FUNCTION_BLOCK "G303M_Code"
TITLE =G303M LOUVER AIR HEATER KILN 2
//COPYRIGHT:    (C) 2009  BUHLER AG, CH-9240 UZWIL, SWITZERLAND
//
//PRODUCT:      WinCoS_BIW01_09
//
//TITLE:        LOUVER AIR HEATER KILN 2
//                Machine group control
//                Maschinengruppensteuerung
//
//--------------------------------------------------------------------------------
//
//IDENT:        AUTHOR:             DEPT:                              DATE:
//
//P01_FB403.2.0 M.Wedler            AEB41                              27.Apr.2010
//             2nd Release
//P01_FB403.1.0 K.Renz              CSB41                              08.Okt.2009
//             1st Release
//
//--------------------------------------------------------------------------------
//
//PURPOSE:
//
//MANUAL :
//
//RESTRICTIONS:
//
//--------------------------------------------------------------------------------
AUTHOR : KR
FAMILY : USW
VERSION : 9.9


VAR
  Gr : "GCS7_GrpCtrlSub";	//Standard interface to group
  InOutValue1 : DINT ;	//Data for user
  InOutValue2 : DINT ;	//Data for user
  OutWayConflict : BOOL ;	//Data for user
  OutSelectionOk : BOOL ;	//Data for user
  CmdNewValue : BOOL ;	//Data for user
  CmdNewJob : BOOL ;	//Data for user
  OutCodeOK : BOOL ;	//Data for user
  InEndOfJob : BOOL ;	//Data for user
  staWayOk : BOOL ;	//Data for user
  EdgeStartRelease : BOOL ;	//Data for user
  USW8 : BOOL ;	//Data for user
  USW9 : BOOL ;	//Data for user
  USW10 : BOOL ;	//Data for user
  USW11 : BOOL ;	//Data for user
  USW12 : BOOL ;	//Data for user
  USW13 : BOOL ;	//Data for user
  USW14 : BOOL ;	//Data for user
  USW15 : BOOL ;	//Data for user
  A_3240_MXZ11 : "GCS7_E_ValveControl4Pos";	// VLS4Ctrl
  A_3240_MXZ11I1 : "GCS7_E_DigInput";	// DigInpCont
  A_3240_MXZ11I11 : "GCS7_E_DigInput";	// DigInpCont
  A_3240_MXZ11I2 : "GCS7_E_DigInput";	// DigInpCont
  A_3240_MXZ11I22 : "GCS7_E_DigInput";	// DigInpCont
  A_3241_MXZ11 : "GCS7_E_ValveControl4Pos";	// VLS4Ctrl
  A_3241_MXZ11I1 : "GCS7_E_DigInput";	// DigInpCont
  A_3241_MXZ11I11 : "GCS7_E_DigInput";	// DigInpCont
  A_3241_MXZ11I2 : "GCS7_E_DigInput";	// DigInpCont
  A_3241_MXZ11I22 : "GCS7_E_DigInput";	// DigInpCont
END_VAR
VAR_TEMP
  tmpEnable : BOOL ;
  tmpFlag : BOOL ;
  tmpCmdNext : BOOL ;
  tmpLocal : BOOL ;
  tmpAspOk : BOOL ;
  tmpHWStop : BOOL ;
  tmpInstanzDBNo : INT ;
END_VAR
BEGIN
NETWORK
TITLE =



NETWORK
TITLE =Read command from group control
//Parameter
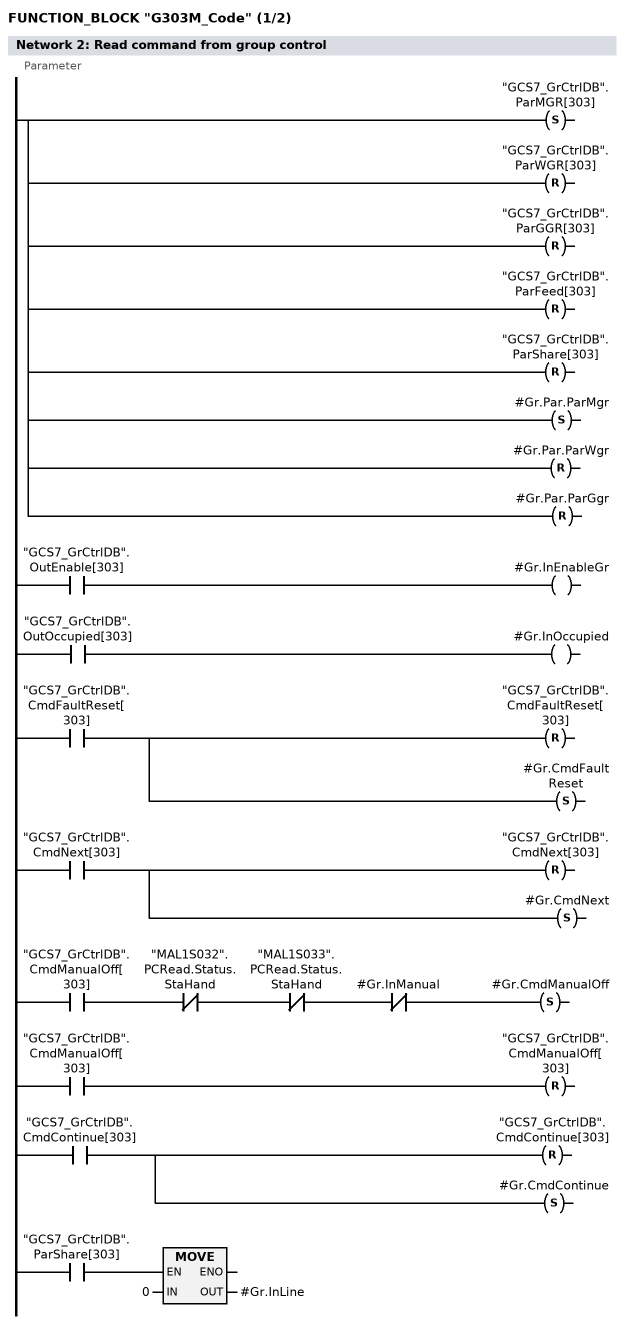
      SET   ;
      S     "GCS7_GrCtrlDB".ParMGR[303];
      R     "GCS7_GrCtrlDB".ParWGR[303];
      R     "GCS7_GrCtrlDB".ParGGR[303];
      R     "GCS7_GrCtrlDB".ParFeed[303];
      R     "GCS7_GrCtrlDB".ParShare[303];
      S     #Gr.Par.ParMgr;
      R     #Gr.Par.ParWgr;
      R     #Gr.Par.ParGgr;
//Command
      U     "GCS7_GrCtrlDB".OutEnable[303];
      =     #Gr.InEnableGr;
      U     "GCS7_GrCtrlDB".OutOccupied[303];
      =     #Gr.InOccupied;
      U     "GCS7_GrCtrlDB".CmdFaultReset[303];
      R     "GCS7_GrCtrlDB".CmdFaultReset[303];
      S     #Gr.CmdFaultReset;
      U     "GCS7_GrCtrlDB".CmdNext[303];
      R     "GCS7_GrCtrlDB".CmdNext[303];
      S     #Gr.CmdNext;

      U     "GCS7_GrCtrlDB".CmdManualOff[303];
      UN    "MAL1S032".PCRead.Status.StaHand;
      UN    "MAL1S033".PCRead.Status.StaHand;
      UN    #Gr.InManual;
      S     #Gr.CmdManualOff;
      U     "GCS7_GrCtrlDB".CmdManualOff[303];
      R     "GCS7_GrCtrlDB".CmdManualOff[303];

//      U     "GCS7_GrCtrlDB".CmdManualOff[303]
//      O     "GCS7_GrCtrlDB".OutOccupied[303]
//      R     "GCS7_GrCtrlDB".CmdManualOff[303]
//      S     #Gr.CmdManualOff

      U     "GCS7_GrCtrlDB".CmdContinue[303];
      R     "GCS7_GrCtrlDB".CmdContinue[303];
      S     #Gr.CmdContinue;
//Init Line Number
      U     "GCS7_GrCtrlDB".ParShare[303];
      SPBN  WE00;
      L     0;
      T     #Gr.InLine;
WE00: NOP   0;
NETWORK
TITLE =Call Methode Control
// 1. Handle Interface PCControl
// 2. Prepare mode --> ModePassive,ModeActive,ModeIdling
// 3. Reset global flags of the group
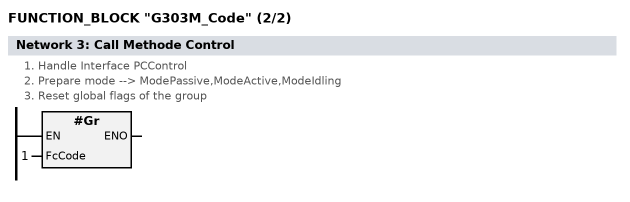
      CALL #Gr (
           FcCode                   := 1);
NETWORK
TITLE =Restart Idling Time

      L     #Gr.Par.ParIdling;
      L     2;
      >=I   ;
      SPB   IdTm;
      T     #Gr.Par.ParIdling;
IdTm: NOP   0;
      U     #A_3240_MXZ11.StNoPosition;
      O     #A_3241_MXZ11.StNoPosition;
      UN    #Gr.InOccupied;
      S     #Gr.CmdRestartIdling;
NETWORK
TITLE =Prepare global flags



NETWORK
TITLE =Set Pattern (Target position)

      L     "MAL1S033Par".Ilo.ILOMode;
      L     5;
      ==I   ;
      U     #Gr.InManual;
      SPBN  M062;
      L     1000;
      T     #A_3240_MXZ11.InPositionMiddle; // setpoint element
      T     #A_3241_MXZ11.InPositionMiddle; // setpoint element
      SPA   M060;
M062: NOP   0;
// setpoint louver air heater
      U     "MAL1S033Par".Par.FlagProcess.ProcessActive;
      UN    "MAL1S033Par".Par.FlagProcess.Cooling_Activ;
      O(    ;
      U     "MAL1S033Par".Par.FlagProcess.Cooling_Activ;
      UN    "G298M".A_3250_MXZ11.StHN;
      UN    "G298M".A_3251_MXZ11.StHN;
      UN    "G298M".A_3252_MXZ11.StHN;
      UN    "G298M".A_3253_MXZ11.StHN;
      )     ;
      SPBN  M061;
      L     1000;
      T     #A_3240_MXZ11.InPositionMiddle; // setpoint element
      T     #A_3241_MXZ11.InPositionMiddle; // setpoint element
M061: NOP   0;
      U(    ;
      U     "MAL1S033Par".Par.FlagProcess.ProcessEnd;
      ON    "MAL1S033Par".Par.FlagProcess.ProcessActive;
      )     ;
      SPBN  M060;
      L     0;
      T     #A_3240_MXZ11.InPositionMiddle; // setpoint element
      T     #A_3241_MXZ11.InPositionMiddle; // setpoint element
M060: NOP   0;

NETWORK
TITLE =Interlocking WayOk



NETWORK
TITLE =Interlocking Autostart

      CLR   ;
      R     #Gr.OutAutostart;
NETWORK
TITLE =Interlocking Enable
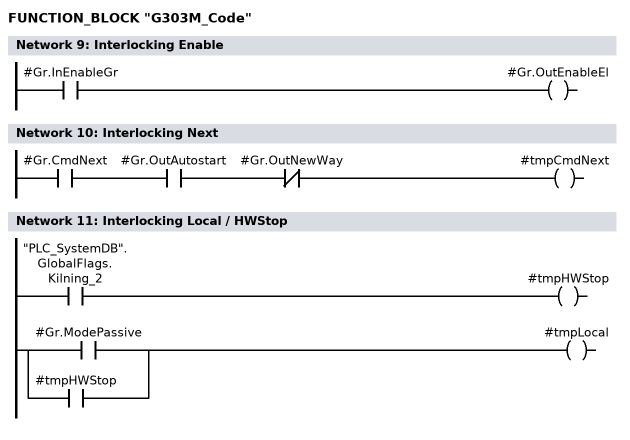

      U     #Gr.InEnableGr;
      =     #Gr.OutEnableEl;

NETWORK
TITLE =Interlocking Next

      U     #Gr.CmdNext;
      U     #Gr.OutAutostart;
      UN    #Gr.OutNewWay;
      =     #tmpCmdNext;

NETWORK
TITLE =Interlocking Local / HWStop

      U     "PLC_SystemDB".GlobalFlags.Kilning_2;
      =     #tmpHWStop;

      U     #Gr.ModePassive;
      O     #tmpHWStop;
      =     #tmpLocal;

NETWORK
TITLE ==A-3240-MXZ11 : LOUVER-AIR ON DOOR FOR RECYCLE AIR 1

      NOP   0;
//-InLocal---
      U(    ;
      U     #tmpLocal;
//      U     #A_3240_MXZ11I11.StTrue
      U     #A_3240_MXZ11.StLN;
      O     ;
      U     #Gr.InManual;
      UN    #Gr.InOutAutostartMan;
      )     ;
      =     #A_3240_MXZ11.InLocal;
//
//-Interlocking---
      U     #A_3240_MXZ11.Par.ParManual;
      U     #A_3240_MXZ11.InManual;
      SPB   man1;
      U(    ;
      UN    #Gr.InOccupied;
      UN    #Gr.InManual;
      )     ;
      O(    ;
      L     0;
      L     #A_3240_MXZ11.InPositionMiddle; // setpoint element
      ==I   ;
      )     ;
      U(    ;
      U     #Gr.InManual;
      U     #Gr.InOutAutostartMan;
      ON    #Gr.InManual;
      )     ;
// Function Added, to get shure always closed in passive state
//      U     #Gr.OutEnableEl
      U(    ;
      U     #Gr.OutEnableEl;
      O     ;
      UN    #Gr.InOccupied;
      UN    #Gr.InManual;
      UN    #A_3240_MXZ11.InLocal;
      )     ;
      =     #A_3240_MXZ11.InLN;

      U(    ;
      L     #A_3240_MXZ11.InPositionMiddle; // setpoint element
      L     0;
      >I    ;
      )     ;
      U(    ;
      L     #A_3240_MXZ11.InPositionMiddle; // setpoint element
      L     1000; // 100,0%
      <I    ;
      )     ;
      U(    ;
      U     #Gr.InManual;
      U     #Gr.InOutAutostartMan;
      ON    #Gr.InManual;
      )     ;
      U     #Gr.OutEnableEl;
      S     #A_3240_MXZ11.CmdMiddle1;

      CLR   ;
      S     #A_3240_MXZ11.CmdMiddle2;

      U(    ;
      L     #A_3240_MXZ11.InPositionMiddle; // setpoint element
      L     1000; // 100,0%
      >=I   ;
      )     ;
      U(    ;
      U     #Gr.InManual;
      U     #Gr.InOutAutostartMan;
      ON    #Gr.InManual;
      )     ;
      U     #Gr.OutEnableEl;
      S     #A_3240_MXZ11.CmdHN;
man1: NOP   0;
//
//-Read inputs---
      U     "A_3240_BZS14_I1";
      =     #A_3240_MXZ11.InpLN;
      CLR   ;
      =     #A_3240_MXZ11.InpMiddle1;
      U     "A_3240_BZS15_I1";
      =     #A_3240_MXZ11.InpHN;
      U     "PLC_SystemDB".GlobalFlags.Kilning_2;
      =     #A_3240_MXZ11.InHWStop;
      U     "PLC_DPInfo".Master[1].SlavesError[101];
      =     #A_3240_MXZ11.InDPFault;
//
//-Set Parameters---
//
//-Call object control---
      CALL #A_3240_MXZ11 ;
//
//-Write outputs---
      U     #A_3240_MXZ11.OutpLN;
      =     "A_3240_MXZ11_O1";
      U     #A_3240_MXZ11.OutpHN;
      =     "A_3240_MXZ11_O2";
NETWORK
TITLE ==A-3240-MXZ11I1 : LOUVER-AIR ON DOOR FOR RECYCLE AIR 1 CLOSING

      NOP   0;
//-InLocal---
      U     #tmpLocal;
      SET   ;
      =     #A_3240_MXZ11I1.InLocal;
//
//-Monitoring---
      U     #A_3240_MXZ11.OutpLN; // closing
      =     #A_3240_MXZ11I1.InMonTrue;
      CLR   ;
      =     #A_3240_MXZ11I1.InMonFalse;
//
//-PreAlarm---
      CLR   ;
      =     #A_3240_MXZ11I1.InPreAlarmTrue;
      CLR   ;
      =     #A_3240_MXZ11I1.InPreAlarmFalse;
//
//-Additional commands---
//      CLR
//      S     #A_3240_MXZ11I1.CmdRunTimeOutTime
//
//-Read inputs---
      U     "A_3240_MXZ11_I1";
      =     #A_3240_MXZ11I1.InpTrue;
      U     "PLC_SystemDB".GlobalFlags.Kilning_2;
      =     #A_3240_MXZ11I1.InHWStop;
      U     "PLC_DPInfo".Master[1].SlavesError[101];
      =     #A_3240_MXZ11I1.InDPFault;
//
//-Set Parameters---
//
//-Call object control---
      CALL #A_3240_MXZ11I1 ;
//
//-Write outputs---
NETWORK
TITLE ==A-3240-MXZ11I11 : LOUVER-AIR ON DOOR FOR RECYCLE AIR 1 CLOSED

      NOP   0;
//-InLocal---
      U     #tmpLocal;
      =     #A_3240_MXZ11I11.InLocal;
//
//-Monitoring---
      CLR   ;
      =     #A_3240_MXZ11I11.InMonTrue;
      CLR   ;
      =     #A_3240_MXZ11I11.InMonFalse;
//
//-PreAlarm---
      CLR   ;
      =     #A_3240_MXZ11I11.InPreAlarmTrue;
      CLR   ;
      =     #A_3240_MXZ11I11.InPreAlarmFalse;
//
//-Additional commands---
//      CLR
//      S     #A_3240_MXZ11I11.CmdRunTimeOutTime
//
//-Read inputs---
      U     "A_3240_MXZ11_I1";
      =     #A_3240_MXZ11I11.InpTrue;
      U     "PLC_SystemDB".GlobalFlags.Kilning_2;
      =     #A_3240_MXZ11I11.InHWStop;
      U     "PLC_DPInfo".Master[1].SlavesError[101];
      =     #A_3240_MXZ11I11.InDPFault;
//
//-Set Parameters---
//
//-Call object control---
      CALL #A_3240_MXZ11I11 ;
//
//-Write outputs---
NETWORK
TITLE ==A-3240-MXZ11I2 : LOUVER-AIR ON DOOR FOR RECYCLE AIR 1 OPENING

      NOP   0;
//-InLocal---
      U     #tmpLocal;
      SET   ;
      =     #A_3240_MXZ11I2.InLocal;
//
//-Monitoring---
      U     #A_3240_MXZ11.OutpHN; // opening
      =     #A_3240_MXZ11I2.InMonTrue;
      CLR   ;
      =     #A_3240_MXZ11I2.InMonFalse;
//
//-PreAlarm---
      CLR   ;
      =     #A_3240_MXZ11I2.InPreAlarmTrue;
      CLR   ;
      =     #A_3240_MXZ11I2.InPreAlarmFalse;
//
//-Additional commands---
//      CLR
//      S     #A_3240_MXZ11I2.CmdRunTimeOutTime
//
//-Read inputs---
      U     "A_3240_MXZ11_I2";
      =     #A_3240_MXZ11I2.InpTrue;
      U     "PLC_SystemDB".GlobalFlags.Kilning_2;
      =     #A_3240_MXZ11I2.InHWStop;
      U     "PLC_DPInfo".Master[1].SlavesError[101];
      =     #A_3240_MXZ11I2.InDPFault;
//
//-Set Parameters---
//
//-Call object control---
      CALL #A_3240_MXZ11I2 ;
//
//-Write outputs---
NETWORK
TITLE ==A-3240-MXZ11I22 : LOUVER-AIR ON DOOR FOR RECYCLE AIR 1 OPENED

      NOP   0;
//-InLocal---
      U     #tmpLocal;
      =     #A_3240_MXZ11I22.InLocal;
//
//-Monitoring---
      CLR   ;
      =     #A_3240_MXZ11I22.InMonTrue;
      CLR   ;
      =     #A_3240_MXZ11I22.InMonFalse;
//
//-PreAlarm---
      CLR   ;
      =     #A_3240_MXZ11I22.InPreAlarmTrue;
      CLR   ;
      =     #A_3240_MXZ11I22.InPreAlarmFalse;
//
//-Additional commands---
//      CLR
//      S     #A_3240_MXZ11I22.CmdRunTimeOutTime
//
//-Read inputs---
      U     "A_3240_MXZ11_I2";
      =     #A_3240_MXZ11I22.InpTrue;
      U     "PLC_SystemDB".GlobalFlags.Kilning_2;
      =     #A_3240_MXZ11I22.InHWStop;
      U     "PLC_DPInfo".Master[1].SlavesError[101];
      =     #A_3240_MXZ11I22.InDPFault;
//
//-Set Parameters---
//
//-Call object control---
      CALL #A_3240_MXZ11I22 ;
//
//-Write outputs---
NETWORK
TITLE ==A-3241-MXZ11 : LOUVER-AIR ON DOOR FOR RECYCLE AIR 2

      NOP   0;
//-InLocal---
      U(    ;
      U     #tmpLocal;
//      U     #A_3241_MXZ11I11.StTrue
      U     #A_3241_MXZ11.StLN;
      O     ;
      U     #Gr.InManual;
      UN    #Gr.InOutAutostartMan;
      )     ;
      =     #A_3241_MXZ11.InLocal;
//
//-Interlocking---
      U     #A_3241_MXZ11.Par.ParManual;
      U     #A_3241_MXZ11.InManual;
      SPB   man2;
      U(    ;
      UN    #Gr.InOccupied;
      UN    #Gr.InManual;
      )     ;
      O(    ;
      L     0;
      L     #A_3241_MXZ11.InPositionMiddle; // setpoint element
      ==I   ;
      )     ;
      U(    ;
      U     #Gr.InManual;
      U     #Gr.InOutAutostartMan;
      ON    #Gr.InManual;
      )     ;
// Function Added, to get shure always closed in passive state
//      U     #Gr.OutEnableEl
      U(    ;
      U     #Gr.OutEnableEl;
      O     ;
      UN    #Gr.InOccupied;
      UN    #Gr.InManual;
      UN    #A_3241_MXZ11.InLocal;
      )     ;
      =     #A_3241_MXZ11.InLN;

      U(    ;
      L     #A_3241_MXZ11.InPositionMiddle; // setpoint element
      L     0;
      >I    ;
      )     ;
      U(    ;
      L     #A_3241_MXZ11.InPositionMiddle; // setpoint element
      L     1000; // 100,0%
      <I    ;
      )     ;
      U(    ;
      U     #Gr.InManual;
      U     #Gr.InOutAutostartMan;
      ON    #Gr.InManual;
      )     ;
      U     #Gr.OutEnableEl;
      S     #A_3241_MXZ11.CmdMiddle1;

      CLR   ;
      S     #A_3241_MXZ11.CmdMiddle2;

      U(    ;
      L     #A_3241_MXZ11.InPositionMiddle; // setpoint element
      L     1000; // 100,0%
      >=I   ;
      )     ;
      U(    ;
      U     #Gr.InManual;
      U     #Gr.InOutAutostartMan;
      ON    #Gr.InManual;
      )     ;
      U     #Gr.OutEnableEl;
      S     #A_3241_MXZ11.CmdHN;
man2: NOP   0;
//
//-Read inputs---
      U     "A_3241_BZS14_I1";
      =     #A_3241_MXZ11.InpLN;
      CLR   ;
      =     #A_3241_MXZ11.InpMiddle1;
      U     "A_3241_BZS15_I1";
      =     #A_3241_MXZ11.InpHN;
      U     "PLC_SystemDB".GlobalFlags.Kilning_2;
      =     #A_3241_MXZ11.InHWStop;
      U     "PLC_DPInfo".Master[1].SlavesError[101];
      =     #A_3241_MXZ11.InDPFault;
//
//-Set Parameters---
//
//-Call object control---
      CALL #A_3241_MXZ11 ;
//
//-Write outputs---
      U     #A_3241_MXZ11.OutpLN;
      =     "A_3241_MXZ11_O1";
      U     #A_3241_MXZ11.OutpHN;
      =     "A_3241_MXZ11_O2";
NETWORK
TITLE ==A-3241-MXZ11I1 : LOUVER-AIR ON DOOR FOR RECYCLE AIR 2 CLOSING

      NOP   0;
//-InLocal---
      U     #tmpLocal;
      SET   ;
      =     #A_3241_MXZ11I1.InLocal;
//
//-Monitoring---
      U     #A_3241_MXZ11.OutpLN; // closing
      =     #A_3241_MXZ11I1.InMonTrue;
      CLR   ;
      =     #A_3241_MXZ11I1.InMonFalse;
//
//-PreAlarm---
      CLR   ;
      =     #A_3241_MXZ11I1.InPreAlarmTrue;
      CLR   ;
      =     #A_3241_MXZ11I1.InPreAlarmFalse;
//
//-Additional commands---
//      CLR
//      S     #A_3241_MXZ11I1.CmdRunTimeOutTime
//
//-Read inputs---
      U     "A_3241_MXZ11_I1";
      =     #A_3241_MXZ11I1.InpTrue;
      U     "PLC_SystemDB".GlobalFlags.Kilning_2;
      =     #A_3241_MXZ11I1.InHWStop;
      U     "PLC_DPInfo".Master[1].SlavesError[101];
      =     #A_3241_MXZ11I1.InDPFault;
//
//-Set Parameters---
//
//-Call object control---
      CALL #A_3241_MXZ11I1 ;
//
//-Write outputs---
NETWORK
TITLE ==A-3241-MXZ11I11 : LOUVER-AIR ON DOOR FOR RECYCLE AIR 2 CLOSED

      NOP   0;
//-InLocal---
      U     #tmpLocal;
      =     #A_3241_MXZ11I11.InLocal;
//
//-Monitoring---
      CLR   ;
      =     #A_3241_MXZ11I11.InMonTrue;
      CLR   ;
      =     #A_3241_MXZ11I11.InMonFalse;
//
//-PreAlarm---
      CLR   ;
      =     #A_3241_MXZ11I11.InPreAlarmTrue;
      CLR   ;
      =     #A_3241_MXZ11I11.InPreAlarmFalse;
//
//-Additional commands---
//      CLR
//      S     #A_3241_MXZ11I11.CmdRunTimeOutTime
//
//-Read inputs---
      U     "A_3241_MXZ11_I1";
      =     #A_3241_MXZ11I11.InpTrue;
      U     "PLC_SystemDB".GlobalFlags.Kilning_2;
      =     #A_3241_MXZ11I11.InHWStop;
      U     "PLC_DPInfo".Master[1].SlavesError[101];
      =     #A_3241_MXZ11I11.InDPFault;
//
//-Set Parameters---
//
//-Call object control---
      CALL #A_3241_MXZ11I11 ;
//
//-Write outputs---
NETWORK
TITLE ==A-3241-MXZ11I2 : LOUVER-AIR ON DOOR FOR RECYCLE AIR 2 OPENING

      NOP   0;
//-InLocal---
      U     #tmpLocal;
      SET   ;
      =     #A_3241_MXZ11I2.InLocal;
//
//-Monitoring---
      U     #A_3241_MXZ11.OutpHN; // opening
      =     #A_3241_MXZ11I2.InMonTrue;
      CLR   ;
      =     #A_3241_MXZ11I2.InMonFalse;
//
//-PreAlarm---
      CLR   ;
      =     #A_3241_MXZ11I2.InPreAlarmTrue;
      CLR   ;
      =     #A_3241_MXZ11I2.InPreAlarmFalse;
//
//-Additional commands---
//      CLR
//      S     #A_3241_MXZ11I2.CmdRunTimeOutTime
//
//-Read inputs---
      U     "A_3241_MXZ11_I2";
      =     #A_3241_MXZ11I2.InpTrue;
      U     "PLC_SystemDB".GlobalFlags.Kilning_2;
      =     #A_3241_MXZ11I2.InHWStop;
      U     "PLC_DPInfo".Master[1].SlavesError[101];
      =     #A_3241_MXZ11I2.InDPFault;
//
//-Set Parameters---
//
//-Call object control---
      CALL #A_3241_MXZ11I2 ;
//
//-Write outputs---
NETWORK
TITLE ==A-3241-MXZ11I22 : LOUVER-AIR ON DOOR FOR RECYCLE AIR 2 OPENED

      NOP   0;
//-InLocal---
      U     #tmpLocal;
      =     #A_3241_MXZ11I22.InLocal;
//
//-Monitoring---
      CLR   ;
      =     #A_3241_MXZ11I22.InMonTrue;
      CLR   ;
      =     #A_3241_MXZ11I22.InMonFalse;
//
//-PreAlarm---
      CLR   ;
      =     #A_3241_MXZ11I22.InPreAlarmTrue;
      CLR   ;
      =     #A_3241_MXZ11I22.InPreAlarmFalse;
//
//-Additional commands---
//      CLR
//      S     #A_3241_MXZ11I22.CmdRunTimeOutTime
//
//-Read inputs---
      U     "A_3241_MXZ11_I2";
      =     #A_3241_MXZ11I22.InpTrue;
      U     "PLC_SystemDB".GlobalFlags.Kilning_2;
      =     #A_3241_MXZ11I22.InHWStop;
      U     "PLC_DPInfo".Master[1].SlavesError[101];
      =     #A_3241_MXZ11I22.InDPFault;
//
//-Set Parameters---
//
//-Call object control---
      CALL #A_3241_MXZ11I22 ;
//
//-Write outputs---
NETWORK
TITLE =Test Fault
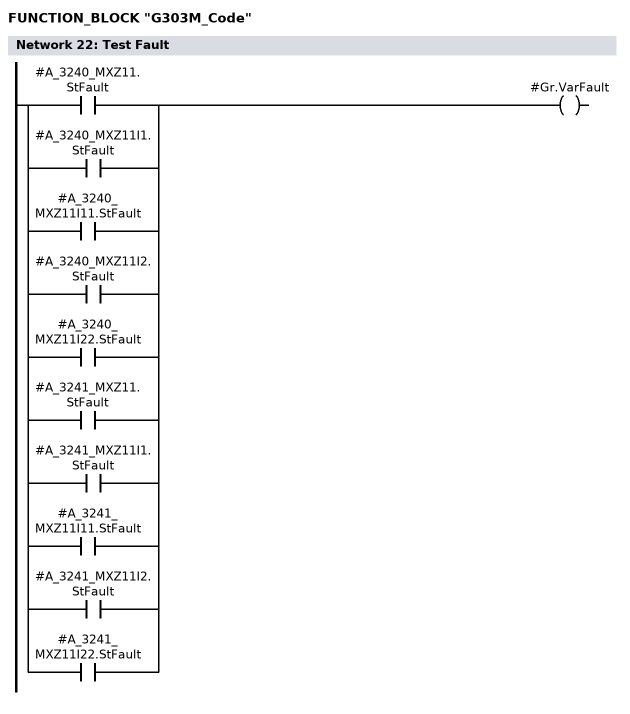

      U     #A_3240_MXZ11.StFault;
      O     #A_3240_MXZ11I1.StFault;
      O     #A_3240_MXZ11I11.StFault;
      O     #A_3240_MXZ11I2.StFault;
      O     #A_3240_MXZ11I22.StFault;
      O     #A_3241_MXZ11.StFault;
      O     #A_3241_MXZ11I1.StFault;
      O     #A_3241_MXZ11I11.StFault;
      O     #A_3241_MXZ11I2.StFault;
      O     #A_3241_MXZ11I22.StFault;
      =     #Gr.VarFault;
NETWORK
TITLE =Test Warning

      CLR   ;
      =     #Gr.OutWarning;
NETWORK
TITLE =Test Stopped
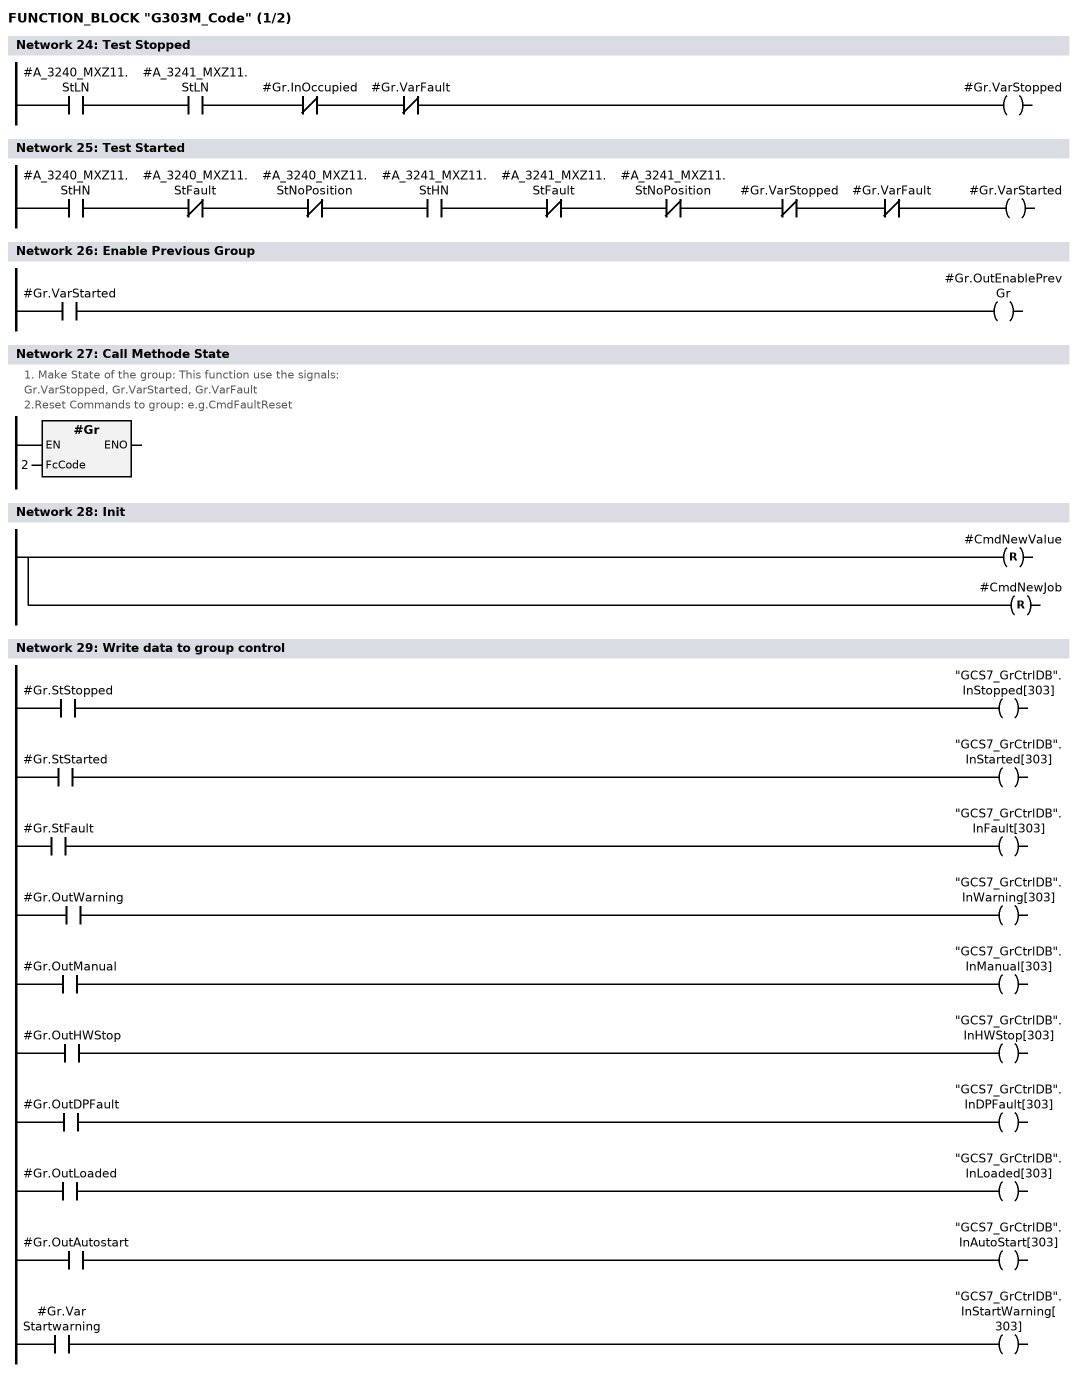

      U     #A_3240_MXZ11.StLN;
      U     #A_3241_MXZ11.StLN;
      UN    #Gr.InOccupied;
      UN    #Gr.VarFault;
      =     #Gr.VarStopped;
NETWORK
TITLE =Test Started

      U     #A_3240_MXZ11.StHN;
      UN    #A_3240_MXZ11.StFault;
      UN    #A_3240_MXZ11.StNoPosition;
      U     #A_3241_MXZ11.StHN;
      UN    #A_3241_MXZ11.StFault;
      UN    #A_3241_MXZ11.StNoPosition;
      UN    #Gr.VarStopped;
      UN    #Gr.VarFault;
      =     #Gr.VarStarted;
NETWORK
TITLE =Enable Previous Group

      U     #Gr.VarStarted;
      =     #Gr.OutEnablePrevGr;
NETWORK
TITLE =Call Methode State
//1. Make State of the group: This function use the signals:
//        Gr.VarStopped, Gr.VarStarted, Gr.VarFault
//2.Reset Commands to group: e.g.CmdFaultReset
      CALL #Gr (
           FcCode                   := 2);
NETWORK
TITLE =Init

      SET   ;
      R     #CmdNewValue;
      R     #CmdNewJob;
NETWORK
TITLE =Write data to group control

      U     #Gr.StStopped;
      =     "GCS7_GrCtrlDB".InStopped[303];
      U     #Gr.StStarted;
      =     "GCS7_GrCtrlDB".InStarted[303];
      U     #Gr.StFault;
      =     "GCS7_GrCtrlDB".InFault[303];
      U     #Gr.OutWarning;
      =     "GCS7_GrCtrlDB".InWarning[303];
      U     #Gr.OutManual;
      =     "GCS7_GrCtrlDB".InManual[303];
      U     #Gr.OutHWStop;
      =     "GCS7_GrCtrlDB".InHWStop[303];
      U     #Gr.OutDPFault;
      =     "GCS7_GrCtrlDB".InDPFault[303];
      U     #Gr.OutLoaded;
      =     "GCS7_GrCtrlDB".InLoaded[303];
      U     #Gr.OutAutostart;
      =     "GCS7_GrCtrlDB".InAutoStart[303];
      U     #Gr.VarStartwarning;
      =     "GCS7_GrCtrlDB".InStartWarning[303];
NETWORK
TITLE =End of block
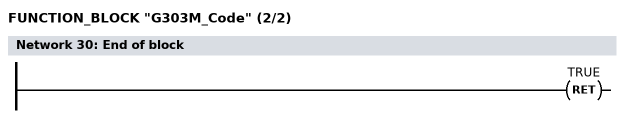

      BE    ;

END_FUNCTION_BLOCK

